(* IEC 61131-3 sources: AXOpen/src/template.axolibrary/ctrl/src/TemplateComponent (part 3) *)

                    IF TRUE THEN
                        THIS.CallTimers(FALSE);
                        _progress := 388;
                    END_IF;
                END_IF;

                IF _progress = 388 THEN                                                                                     // TemplateTask_20steps_2 running: , add_the_detailed_description_of_the_current_action_9
                    IF _infoTimer.output THEN
                        TaskMessenger.Activate( UINT#588, eAxoMessageCategory#Warning);
                        Status.Error.Id :=      UINT#588;
                    END_IF;

                    IF TRUE THEN
                        THIS.CallTimers(FALSE);
                        _progress := 389;
                    END_IF;
                END_IF;

                IF _progress = 389 THEN                                                                                     // TemplateTask_20steps_2 running: , add_the_detailed_description_of_the_current_action_10
                    IF _infoTimer.output THEN
                        TaskMessenger.Activate( UINT#589, eAxoMessageCategory#Warning);
                        Status.Error.Id :=      UINT#589;
                    END_IF;

                    IF TRUE THEN
                        THIS.CallTimers(FALSE);
                        _progress := 390;
                    END_IF;
                END_IF;

                IF _progress = 390 THEN                                                                                     // TemplateTask_20steps_2 running: , add_the_detailed_description_of_the_current_action_11
                    IF _infoTimer.output THEN
                        TaskMessenger.Activate( UINT#590, eAxoMessageCategory#Warning);
                        Status.Error.Id :=      UINT#590;
                    END_IF;

                    IF TRUE THEN
                        THIS.CallTimers(FALSE);
                        _progress := 391;
                    END_IF;
                END_IF;

                IF _progress = 391 THEN                                                                                     // TemplateTask_20steps_2 running: , add_the_detailed_description_of_the_current_action_12
                    IF _infoTimer.output THEN
                        TaskMessenger.Activate( UINT#591, eAxoMessageCategory#Warning);
                        Status.Error.Id :=      UINT#591;
                    END_IF;

                    IF TRUE THEN
                        THIS.CallTimers(FALSE);
                        _progress := 392;
                    END_IF;
                END_IF;

                IF _progress = 392 THEN                                                                                     // TemplateTask_20steps_2 running: , add_the_detailed_description_of_the_current_action_13
                    IF _infoTimer.output THEN
                        TaskMessenger.Activate( UINT#592, eAxoMessageCategory#Warning);
                        Status.Error.Id :=      UINT#592;
                    END_IF;;

                    IF TRUE THEN
                        THIS.CallTimers(FALSE);
                        _progress := 393;
                    END_IF;
                END_IF;

                IF _progress = 393 THEN                                                                                     // TemplateTask_20steps_2 running: , add_the_detailed_description_of_the_current_action_14
                    IF _infoTimer.output THEN
                        TaskMessenger.Activate( UINT#593, eAxoMessageCategory#Warning);
                        Status.Error.Id :=      UINT#593;
                    END_IF;

                    IF TRUE THEN
                        THIS.CallTimers(FALSE);
                        _progress := 394;
                    END_IF;
                END_IF;

                IF _progress = 394 THEN                                                                                     // TemplateTask_20steps_2 running: , add_the_detailed_description_of_the_current_action_15
                    IF _infoTimer.output THEN
                        TaskMessenger.Activate( UINT#594, eAxoMessageCategory#Warning);
                        Status.Error.Id :=      UINT#594;
                    END_IF;

                    IF TRUE THEN
                        THIS.CallTimers(FALSE);
                        _progress := 395;
                    END_IF;
                END_IF;

                IF _progress = 395 THEN                                                                                     // TemplateTask_20steps_2 running: , add_the_detailed_description_of_the_current_action_16
                    IF _infoTimer.output THEN
                        TaskMessenger.Activate( UINT#595, eAxoMessageCategory#Warning);
                        Status.Error.Id :=      UINT#595;
                    END_IF;

                    IF TRUE THEN
                        THIS.CallTimers(FALSE);
                        _progress := 396;
                    END_IF;
                END_IF;

                IF _progress = 396 THEN                                                                                     // TemplateTask_20steps_2 running: , add_the_detailed_description_of_the_current_action_17
                    IF _infoTimer.output THEN
                        TaskMessenger.Activate( UINT#596, eAxoMessageCategory#Warning);
                        Status.Error.Id :=      UINT#596;
                    END_IF;

                    IF TRUE THEN
                        THIS.CallTimers(FALSE);
                        _progress := 397;
                    END_IF;
                END_IF;

                IF _progress = 397 THEN                                                                                     // TemplateTask_20steps_2 running: , add_the_detailed_description_of_the_current_action_18
                    IF _infoTimer.output THEN
                        TaskMessenger.Activate( UINT#597, eAxoMessageCategory#Warning);
                        Status.Error.Id :=      UINT#597;
                    END_IF;

                    IF TRUE THEN
                        THIS.CallTimers(FALSE);
                        _progress := 398;
                    END_IF;
                END_IF;

                IF _progress = 398 THEN                                                                                     // TemplateTask_20steps_2 running: , add_the_detailed_description_of_the_current_action_19
                    IF _infoTimer.output THEN
                        TaskMessenger.Activate( UINT#598, eAxoMessageCategory#Warning);
                        Status.Error.Id :=      UINT#598;
                    END_IF;

                    IF TRUE THEN
                        THIS.CallTimers(FALSE);
                        _progress := 399;
                    END_IF;
                END_IF;

                IF _progress = 399 THEN                                                                                     // TemplateTask_20steps_2 running: , add_the_detailed_description_of_the_current_action_20
                    TemplateTask_20steps_2.DoneWhen(TRUE);
                    _progress := 0;
                END_IF;

                THIS.CallTimers(TRUE);
                TemplateTask_20steps_2.ThrowWhen(_errorTimer.output);
                Status.Action.Id := TO_UINT(_progress);
                TemplateTask_20steps_2.ThrowWhen(TemplateTask_20steps_2.Duration >= Config.TaskTimeout AND Config.TaskTimeout > T#0s ,'TemplateTask_20steps_2 timeout.');
            END_IF;
            IF TemplateTask_20steps_2.DoneReached() THEN
                Status.Action.Id :=  UINT#181;
                Status.Error.Id :=  UINT#0;
            ELSIF TemplateTask_20steps_2.ErrorOccured() THEN
                Status.Action.Id :=  UINT#10080;
                Status.Error.Id  :=  UINT#10080;
            ELSIF TemplateTask_20steps_2.AbortTriggered()THEN
                Status.Action.Id :=  UINT#10081;
                Status.Error.Id  :=  UINT#10081;
            END_IF;
            Messenger.ActivateOnCondition(ULINT#10080,TemplateTask_20steps_2.HasError(), eAxoMessageCategory#Error);
            Messenger.ActivateOnCondition(ULINT#10081,TemplateTask_20steps_2.IsAborted(), eAxoMessageCategory#Error);
            Messenger.ActivateOnCondition(ULINT#182,TemplateTask_20steps_2.RestoreTriggered() , eAxoMessageCategory#Error);
            IF TemplateTask_20steps_2.RestoreTriggered() AND _progress >= 380 AND _progress <= 399  THEN
                Status.Action.Id :=  UINT#182;
                _progress := 0;
            END_IF;
            //**************************************************

            //*************TemplateTask_20steps_3***************
            TemplateTask_20steps_3.SetIsDisabled(FALSE);
            IF TemplateTask_20steps_3.StartTriggered() THEN
                Status.Action.Id :=  UINT#200;
            END_IF;
            Messenger.ActivateOnCondition(ULINT#200,TemplateTask_20steps_3.IsBusy(), eAxoMessageCategory#Info);
            Messenger.ActivateOnCondition(ULINT#201,TemplateTask_20steps_3.IsDone(), eAxoMessageCategory#Info);
            IF TemplateTask_20steps_3.Execute(THIS) THEN
                IF _progress = 0 THEN
                    Status.Error.Id := UINT#0;
                    TaskMessenger.Restore();
                    THIS.CallTimers(FALSE);
                    _progress := 400;
                END_IF;

                IF _progress = 400 THEN                                                                                     // TemplateTask_20steps_3 running: , add_the_detailed_description_of_the_current_action_1
                    IF _infoTimer.output THEN
                        TaskMessenger.Activate( UINT#600, eAxoMessageCategory#Warning);
                        Status.Error.Id :=      UINT#600;
                    END_IF;

                    IF TRUE THEN
                        THIS.CallTimers(FALSE);
                        _progress := 401;
                    END_IF;
                END_IF;

                IF _progress = 401 THEN                                                                                     // TemplateTask_20steps_3 running: , add_the_detailed_description_of_the_current_action_2
                    IF _infoTimer.output THEN
                        TaskMessenger.Activate( UINT#601, eAxoMessageCategory#Warning);
                        Status.Error.Id :=      UINT#601;
                    END_IF;

                    IF TRUE THEN
                        THIS.CallTimers(FALSE);
                        _progress := 402;
                    END_IF;
                END_IF;

                IF _progress = 402 THEN                                                                                     // TemplateTask_20steps_3 running: , add_the_detailed_description_of_the_current_action_3
                    IF _infoTimer.output THEN
                        TaskMessenger.Activate( UINT#602, eAxoMessageCategory#Warning);
                        Status.Error.Id :=      UINT#602;
                    END_IF;

                    IF TRUE THEN
                        THIS.CallTimers(FALSE);
                        _progress := 403;
                    END_IF;
                END_IF;

                IF _progress = 403 THEN                                                                                     // TemplateTask_20steps_3 running: , add_the_detailed_description_of_the_current_action_4
                    IF _infoTimer.output THEN
                        TaskMessenger.Activate( UINT#603, eAxoMessageCategory#Warning);
                        Status.Error.Id :=      UINT#603;
                    END_IF;

                    IF TRUE THEN
                        THIS.CallTimers(FALSE);
                        _progress := 404;
                    END_IF;
                END_IF;

                IF _progress = 404 THEN                                                                                     // TemplateTask_20steps_3 running: , add_the_detailed_description_of_the_current_action_5
                    IF _infoTimer.output THEN
                        TaskMessenger.Activate( UINT#604, eAxoMessageCategory#Warning);
                        Status.Error.Id :=      UINT#604;
                    END_IF;

                    IF TRUE THEN
                        THIS.CallTimers(FALSE);
                        _progress := 405;
                    END_IF;
                END_IF;

                IF _progress = 405 THEN                                                                                     // TemplateTask_20steps_3 running: , add_the_detailed_description_of_the_current_action_6
                    IF _infoTimer.output THEN
                        TaskMessenger.Activate( UINT#605, eAxoMessageCategory#Warning);
                        Status.Error.Id :=      UINT#605;
                    END_IF;

                    IF TRUE THEN
                        THIS.CallTimers(FALSE);
                        _progress := 406;
                    END_IF;
                END_IF;

                IF _progress = 406 THEN                                                                                     // TemplateTask_20steps_3 running: , add_the_detailed_description_of_the_current_action_7
                    IF _infoTimer.output THEN
                        TaskMessenger.Activate( UINT#606, eAxoMessageCategory#Warning);
                        Status.Error.Id :=      UINT#606;
                    END_IF;

                    IF TRUE THEN
                        THIS.CallTimers(FALSE);
                        _progress := 407;
                    END_IF;
                END_IF;

                IF _progress = 407 THEN                                                                                     // TemplateTask_20steps_3 running: , add_the_detailed_description_of_the_current_action_8
                    IF _infoTimer.output THEN
                        TaskMessenger.Activate( UINT#607, eAxoMessageCategory#Warning);
                        Status.Error.Id :=      UINT#607;
                    END_IF;

                    IF TRUE THEN
                        THIS.CallTimers(FALSE);
                        _progress := 408;
                    END_IF;
                END_IF;

                IF _progress = 408 THEN                                                                                     // TemplateTask_20steps_3 running: , add_the_detailed_description_of_the_current_action_9
                    IF _infoTimer.output THEN
                        TaskMessenger.Activate( UINT#608, eAxoMessageCategory#Warning);
                        Status.Error.Id :=      UINT#608;
                    END_IF;

                    IF TRUE THEN
                        THIS.CallTimers(FALSE);
                        _progress := 409;
                    END_IF;
                END_IF;

                IF _progress = 409 THEN                                                                                     // TemplateTask_20steps_3 running: , add_the_detailed_description_of_the_current_action_10
                    IF _infoTimer.output THEN
                        TaskMessenger.Activate( UINT#609, eAxoMessageCategory#Warning);
                        Status.Error.Id :=      UINT#609;
                    END_IF;

                    IF TRUE THEN
                        THIS.CallTimers(FALSE);
                        _progress := 410;
                    END_IF;
                END_IF;

                IF _progress = 410 THEN                                                                                     // TemplateTask_20steps_3 running: , add_the_detailed_description_of_the_current_action_11
                    IF _infoTimer.output THEN
                        TaskMessenger.Activate( UINT#610, eAxoMessageCategory#Warning);
                        Status.Error.Id :=      UINT#610;
                    END_IF;

                    IF TRUE THEN
                        THIS.CallTimers(FALSE);
                        _progress := 411;
                    END_IF;
                END_IF;

                IF _progress = 411 THEN                                                                                     // TemplateTask_20steps_3 running: , add_the_detailed_description_of_the_current_action_12
                    IF _infoTimer.output THEN
                        TaskMessenger.Activate( UINT#611, eAxoMessageCategory#Warning);
                        Status.Error.Id :=      UINT#611;
                    END_IF;

                    IF TRUE THEN
                        THIS.CallTimers(FALSE);
                        _progress := 412;
                    END_IF;
                END_IF;

                IF _progress = 412 THEN                                                                                     // TemplateTask_20steps_3 running: , add_the_detailed_description_of_the_current_action_13
                    IF _infoTimer.output THEN
                        TaskMessenger.Activate( UINT#612, eAxoMessageCategory#Warning);
                        Status.Error.Id :=      UINT#612;
                    END_IF;

                    IF TRUE THEN
                        THIS.CallTimers(FALSE);
                        _progress := 413;
                    END_IF;
                END_IF;

                IF _progress = 413 THEN                                                                                     // TemplateTask_20steps_3 running: , add_the_detailed_description_of_the_current_action_14
                    IF _infoTimer.output THEN
                        TaskMessenger.Activate( UINT#613, eAxoMessageCategory#Warning);
                        Status.Error.Id :=      UINT#613;
                    END_IF;

                    IF TRUE THEN
                        THIS.CallTimers(FALSE);
                        _progress := 414;
                    END_IF;
                END_IF;

                IF _progress = 414 THEN                                                                                     // TemplateTask_20steps_3 running: , add_the_detailed_description_of_the_current_action_15
                    IF _infoTimer.output THEN
                        TaskMessenger.Activate( UINT#614, eAxoMessageCategory#Warning);
                        Status.Error.Id :=      UINT#614;
                    END_IF;

                    IF TRUE THEN
                        THIS.CallTimers(FALSE);
                        _progress := 415;
                    END_IF;
                END_IF;

                IF _progress = 415 THEN                                                                                     // TemplateTask_20steps_3 running: , add_the_detailed_description_of_the_current_action_16
                    IF _infoTimer.output THEN
                        TaskMessenger.Activate( UINT#615, eAxoMessageCategory#Warning);
                        Status.Error.Id :=      UINT#615;
                    END_IF;

                    IF TRUE THEN
                        THIS.CallTimers(FALSE);
                        _progress := 416;
                    END_IF;
                END_IF;

                IF _progress = 416 THEN                                                                                     // TemplateTask_20steps_3 running: , add_the_detailed_description_of_the_current_action_17
                    IF _infoTimer.output THEN
                        TaskMessenger.Activate( UINT#616, eAxoMessageCategory#Warning);
                        Status.Error.Id :=      UINT#616;
                    END_IF;

                    IF TRUE THEN
                        THIS.CallTimers(FALSE);
                        _progress := 417;
                    END_IF;
                END_IF;

                IF _progress = 417 THEN                                                                                     // TemplateTask_20steps_3 running: , add_the_detailed_description_of_the_current_action_18
                    IF _infoTimer.output THEN
                        TaskMessenger.Activate( UINT#617, eAxoMessageCategory#Warning);
                        Status.Error.Id :=      UINT#617;
                    END_IF;

                    IF TRUE THEN
                        THIS.CallTimers(FALSE);
                        _progress := 418;
                    END_IF;
                END_IF;

                IF _progress = 418 THEN                                                                                     // TemplateTask_20steps_3 running: , add_the_detailed_description_of_the_current_action_19
                    IF _infoTimer.output THEN
                        TaskMessenger.Activate( UINT#618, eAxoMessageCategory#Warning);
                        Status.Error.Id :=      UINT#618;
                    END_IF;

                    IF TRUE THEN
                        THIS.CallTimers(FALSE);
                        _progress := 419;
                    END_IF;
                END_IF;

                IF _progress = 419 THEN                                                                                     // TemplateTask_20steps_3 running: , add_the_detailed_description_of_the_current_action_20
                    TemplateTask_20steps_3.DoneWhen(TRUE);
                    _progress := 0;
                END_IF;

                THIS.CallTimers(TRUE);

                TemplateTask_20steps_3.ThrowWhen(_errorTimer.output);
                Status.Action.Id := TO_UINT(_progress);
                TemplateTask_20steps_3.ThrowWhen(TemplateTask_20steps_3.Duration >= Config.TaskTimeout AND Config.TaskTimeout > T#0s ,'TemplateTask_20steps_3 timeout.');
            END_IF;
            IF TemplateTask_20steps_3.DoneReached() THEN
                Status.Action.Id :=  UINT#201;
                Status.Error.Id :=  UINT#0;
            ELSIF TemplateTask_20steps_3.ErrorOccured() THEN
                Status.Action.Id :=  UINT#10100;
                Status.Error.Id  :=  UINT#10100;
            ELSIF TemplateTask_20steps_3.AbortTriggered()THEN
                Status.Action.Id :=  UINT#10101;
                Status.Error.Id  :=  UINT#10101;
            END_IF;
            Messenger.ActivateOnCondition(ULINT#10100,TemplateTask_20steps_3.HasError(), eAxoMessageCategory#Error);
            Messenger.ActivateOnCondition(ULINT#10101,TemplateTask_20steps_3.IsAborted(), eAxoMessageCategory#Error);
            Messenger.ActivateOnCondition(ULINT#202,TemplateTask_20steps_3.RestoreTriggered() , eAxoMessageCategory#Error);
            IF TemplateTask_20steps_3.RestoreTriggered() AND _progress >= 400 AND _progress <= 419  THEN
                Status.Action.Id :=  UINT#202;
                _progress := 0;
            END_IF;
            //**************************************************

            //*************TemplateTask_20steps_4***************
            TemplateTask_20steps_4.SetIsDisabled(FALSE);
            IF TemplateTask_20steps_4.StartTriggered() THEN
                Status.Action.Id :=  UINT#220;
            END_IF;
            Messenger.ActivateOnCondition(ULINT#220,TemplateTask_20steps_4.IsBusy(), eAxoMessageCategory#Info);
            Messenger.ActivateOnCondition(ULINT#221,TemplateTask_20steps_4.IsDone(), eAxoMessageCategory#Info);
            IF TemplateTask_20steps_4.Execute(THIS) THEN
                IF _progress = 0 THEN
                    Status.Error.Id := UINT#0;
                    TaskMessenger.Restore();
                    THIS.CallTimers(FALSE);
                    _progress := 420;
                END_IF;

                IF _progress = 420 THEN                                                                                     // TemplateTask_20steps_4 running: , add_the_detailed_description_of_the_current_action_1
                    IF _infoTimer.output THEN
                        TaskMessenger.Activate( UINT#620, eAxoMessageCategory#Warning);
                        Status.Error.Id :=      UINT#620;
                    END_IF;

                    IF TRUE THEN
                        THIS.CallTimers(FALSE);
                        _progress := 421;
                    END_IF;
                END_IF;

                IF _progress = 421 THEN                                                                                     // TemplateTask_20steps_4 running: , add_the_detailed_description_of_the_current_action_2
                    IF _infoTimer.output THEN
                        TaskMessenger.Activate( UINT#621, eAxoMessageCategory#Warning);
                        Status.Error.Id :=      UINT#621;
                    END_IF;

                    IF TRUE THEN
                        THIS.CallTimers(FALSE);
                        _progress := 422;
                    END_IF;
                END_IF;

                IF _progress = 422 THEN                                                                                     // TemplateTask_20steps_4 running: , add_the_detailed_description_of_the_current_action_3
                    IF _infoTimer.output THEN
                        TaskMessenger.Activate( UINT#622, eAxoMessageCategory#Warning);
                        Status.Error.Id :=      UINT#622;
                    END_IF;

                    IF TRUE THEN
                        THIS.CallTimers(FALSE);
                        _progress := 423;
                    END_IF;
                END_IF;

                IF _progress = 423 THEN                                                                                     // TemplateTask_20steps_4 running: , add_the_detailed_description_of_the_current_action_4
                    IF _infoTimer.output THEN
                        TaskMessenger.Activate( UINT#623, eAxoMessageCategory#Warning);
                        Status.Error.Id :=      UINT#623;
                    END_IF;

                    IF TRUE THEN
                        THIS.CallTimers(FALSE);
                        _progress := 424;
                    END_IF;
                END_IF;

                IF _progress = 424 THEN                                                                                     // TemplateTask_20steps_4 running: , add_the_detailed_description_of_the_current_action_5
                    IF _infoTimer.output THEN
                        TaskMessenger.Activate( UINT#624, eAxoMessageCategory#Warning);
                        Status.Error.Id :=      UINT#624;
                    END_IF;

                    IF TRUE THEN
                        THIS.CallTimers(FALSE);
                        _progress := 425;
                    END_IF;
                END_IF;

                IF _progress = 425 THEN                                                                                     // TemplateTask_20steps_4 running: , add_the_detailed_description_of_the_current_action_6
                    IF _infoTimer.output THEN
                        TaskMessenger.Activate( UINT#625, eAxoMessageCategory#Warning);
                        Status.Error.Id :=      UINT#625;
                    END_IF;

                    IF TRUE THEN
                        THIS.CallTimers(FALSE);
                        _progress := 426;
                    END_IF;
                END_IF;

                IF _progress = 426 THEN                                                                                     // TemplateTask_20steps_4 running: , add_the_detailed_description_of_the_current_action_7
                    IF _infoTimer.output THEN
                        TaskMessenger.Activate( UINT#626, eAxoMessageCategory#Warning);
                        Status.Error.Id :=      UINT#626;
                    END_IF;

                    IF TRUE THEN
                        THIS.CallTimers(FALSE);
                        _progress := 427;
                    END_IF;
                END_IF;

                IF _progress = 427 THEN                                                                                     // TemplateTask_20steps_4 running: , add_the_detailed_description_of_the_current_action_8
                    IF _infoTimer.output THEN
                        TaskMessenger.Activate( UINT#627, eAxoMessageCategory#Warning);
                        Status.Error.Id :=      UINT#627;
                    END_IF;

                    IF TRUE THEN
                        THIS.CallTimers(FALSE);
                        _progress := 428;
                    END_IF;
                END_IF;

                IF _progress = 428 THEN                                                                                     // TemplateTask_20steps_4 running: , add_the_detailed_description_of_the_current_action_9
                    IF _infoTimer.output THEN
                        TaskMessenger.Activate( UINT#628, eAxoMessageCategory#Warning);
                        Status.Error.Id :=      UINT#628;
                    END_IF;

                    IF TRUE THEN
                        THIS.CallTimers(FALSE);
                        _progress := 429;
                    END_IF;
                END_IF;

                IF _progress = 429 THEN                                                                                     // TemplateTask_20steps_4 running: , add_the_detailed_description_of_the_current_action_10
                    IF _infoTimer.output THEN
                        TaskMessenger.Activate( UINT#629, eAxoMessageCategory#Warning);
                        Status.Error.Id :=      UINT#629;
                    END_IF;

                    IF TRUE THEN
                        THIS.CallTimers(FALSE);
                        _progress := 430;
                    END_IF;
                END_IF;

                IF _progress = 430 THEN                                                                                     // TemplateTask_20steps_4 running: , add_the_detailed_description_of_the_current_action_11
                    IF _infoTimer.output THEN
                        TaskMessenger.Activate( UINT#630, eAxoMessageCategory#Warning);
                        Status.Error.Id :=      UINT#630;
                    END_IF;

                    IF TRUE THEN
                        THIS.CallTimers(FALSE);
                        _progress := 431;
                    END_IF;
                END_IF;

                IF _progress = 431 THEN                                                                                     // TemplateTask_20steps_4 running: , add_the_detailed_description_of_the_current_action_12
                    IF _infoTimer.output THEN
                        TaskMessenger.Activate( UINT#631, eAxoMessageCategory#Warning);
                        Status.Error.Id :=      UINT#631;
                    END_IF;

                    IF TRUE THEN
                        THIS.CallTimers(FALSE);
                        _progress := 432;
                    END_IF;
                END_IF;

                IF _progress = 432 THEN                                                                                     // TemplateTask_20steps_4 running: , add_the_detailed_description_of_the_current_action_13
                    IF _infoTimer.output THEN
                        TaskMessenger.Activate( UINT#632, eAxoMessageCategory#Warning);
                        Status.Error.Id :=      UINT#632;
                    END_IF;

                    IF TRUE THEN
                        THIS.CallTimers(FALSE);
                        _progress := 433;
                    END_IF;
                END_IF;

                IF _progress = 433 THEN                                                                                     // TemplateTask_20steps_4 running: , add_the_detailed_description_of_the_current_action_14
                    IF _infoTimer.output THEN
                        TaskMessenger.Activate( UINT#633, eAxoMessageCategory#Warning);
                        Status.Error.Id :=      UINT#633;
                    END_IF;

                    IF TRUE THEN
                        THIS.CallTimers(FALSE);
                        _progress := 434;
                    END_IF;
                END_IF;

                IF _progress = 434 THEN                                                                                     // TemplateTask_20steps_4 running: , add_the_detailed_description_of_the_current_action_15
                    IF _infoTimer.output THEN
                        TaskMessenger.Activate( UINT#634, eAxoMessageCategory#Warning);
                        Status.Error.Id :=      UINT#634;
                    END_IF;

                    IF TRUE THEN
                        THIS.CallTimers(FALSE);
                        _progress := 435;
                    END_IF;
                END_IF;

                IF _progress = 435 THEN                                                                                     // TemplateTask_20steps_4 running: , add_the_detailed_description_of_the_current_action_16
                    IF _infoTimer.output THEN
                        TaskMessenger.Activate( UINT#635, eAxoMessageCategory#Warning);
                        Status.Error.Id :=      UINT#635;
                    END_IF;

                    IF TRUE THEN
                        THIS.CallTimers(FALSE);
                        _progress := 436;
                    END_IF;
                END_IF;

                IF _progress = 436 THEN                                                                                     // TemplateTask_20steps_4 running: , add_the_detailed_description_of_the_current_action_17
                    IF _infoTimer.output THEN
                        TaskMessenger.Activate( UINT#636, eAxoMessageCategory#Warning);
                        Status.Error.Id :=      UINT#636;
                    END_IF;

                    IF TRUE THEN
                        THIS.CallTimers(FALSE);
                        _progress := 437;
                    END_IF;
                END_IF;

                IF _progress = 437 THEN                                                                                     // TemplateTask_20steps_4 running: , add_the_detailed_description_of_the_current_action_18
                    IF _infoTimer.output THEN
                        TaskMessenger.Activate( UINT#637, eAxoMessageCategory#Warning);
                        Status.Error.Id :=      UINT#637;
                    END_IF;

                    IF TRUE THEN
                        THIS.CallTimers(FALSE);
                        _progress := 438;
                    END_IF;
                END_IF;

                IF _progress = 438 THEN                                                                                     // TemplateTask_20steps_4 running: , add_the_detailed_description_of_the_current_action_19
                    IF _infoTimer.output THEN
                        TaskMessenger.Activate( UINT#638, eAxoMessageCategory#Warning);
                        Status.Error.Id :=      UINT#638;
                    END_IF;

                    IF TRUE THEN
                        THIS.CallTimers(FALSE);
                        _progress := 439;
                    END_IF;
                END_IF;

                IF _progress = 439 THEN                                                                                     // TemplateTask_20steps_4 running: , add_the_detailed_description_of_the_current_action_20
                    TemplateTask_20steps_4.DoneWhen(TRUE);
                    _progress := 0;
                END_IF;

                THIS.CallTimers(TRUE);

                TemplateTask_20steps_4.ThrowWhen(_errorTimer.output);
                Status.Action.Id := TO_UINT(_progress);
                TemplateTask_20steps_4.ThrowWhen(TemplateTask_20steps_4.Duration >= Config.TaskTimeout AND Config.TaskTimeout > T#0s ,'TemplateTask_20steps_4 timeout.');
            END_IF;
            IF TemplateTask_20steps_4.DoneReached() THEN
                Status.Action.Id :=  UINT#221;
                Status.Error.Id :=  UINT#0;
            ELSIF TemplateTask_20steps_4.ErrorOccured() THEN
                Status.Action.Id :=  UINT#10120;
                Status.Error.Id  :=  UINT#10120;
            ELSIF TemplateTask_20steps_4.AbortTriggered()THEN
                Status.Action.Id :=  UINT#10121;
                Status.Error.Id  :=  UINT#10121;
            END_IF;
            Messenger.ActivateOnCondition(ULINT#10120,TemplateTask_20steps_4.HasError(), eAxoMessageCategory#Error);
            Messenger.ActivateOnCondition(ULINT#10121,TemplateTask_20steps_4.IsAborted(), eAxoMessageCategory#Error);
            Messenger.ActivateOnCondition(ULINT#222,TemplateTask_20steps_4.RestoreTriggered() , eAxoMessageCategory#Error);
            IF TemplateTask_20steps_4.RestoreTriggered() AND _progress >= 420 AND _progress <= 439  THEN
                Status.Action.Id :=  UINT#222;
                _progress := 0;
            END_IF;
            //**************************************************

            //*************TemplateTask_20steps_5***************
            TemplateTask_20steps_5.SetIsDisabled(FALSE);
            IF TemplateTask_20steps_5.StartTriggered() THEN
                Status.Action.Id :=  UINT#240;
            END_IF;
            Messenger.ActivateOnCondition(ULINT#240,TemplateTask_20steps_5.IsBusy(), eAxoMessageCategory#Info);
            Messenger.ActivateOnCondition(ULINT#241,TemplateTask_20steps_5.IsDone(), eAxoMessageCategory#Info);
            IF TemplateTask_20steps_5.Execute(THIS) THEN
                IF _progress = 0 THEN
                    Status.Error.Id := UINT#0;
                    TaskMessenger.Restore();
                    THIS.CallTimers(FALSE);
                    _progress := 440;
                END_IF;

                IF _progress = 440 THEN                                                                                     // TemplateTask_20steps_5 running: , add_the_detailed_description_of_the_current_action_1
                    IF _infoTimer.output THEN
                        TaskMessenger.Activate( UINT#640, eAxoMessageCategory#Warning);
                        Status.Error.Id :=      UINT#640;
                    END_IF;

                    IF TRUE THEN
                        THIS.CallTimers(FALSE);
                        _progress := 441;
                    END_IF;
                END_IF;

                IF _progress = 441 THEN                                                                                     // TemplateTask_20steps_5 running , add_the_detailed_description_of_the_current_action_2
                    IF _infoTimer.output THEN
                        TaskMessenger.Activate( UINT#641, eAxoMessageCategory#Warning);
                        Status.Error.Id :=      UINT#641;
                    END_IF;

                    IF TRUE THEN
                        THIS.CallTimers(FALSE);
                        _progress := 442;
                    END_IF;
                END_IF;

                IF _progress = 442 THEN                                                                                     // TemplateTask_20steps_5 running: , add_the_detailed_description_of_the_current_action_3
                    IF _infoTimer.output THEN
                        TaskMessenger.Activate( UINT#642, eAxoMessageCategory#Warning);
                        Status.Error.Id :=      UINT#642;
                    END_IF;

                    IF TRUE THEN
                        THIS.CallTimers(FALSE);
                        _progress := 443;
                    END_IF;
                END_IF;

                IF _progress = 443 THEN                                                                                     // TemplateTask_20steps_5 running: , add_the_detailed_description_of_the_current_action_4
                    IF _infoTimer.output THEN
                        TaskMessenger.Activate( UINT#643, eAxoMessageCategory#Warning);
                        Status.Error.Id :=      UINT#643;
                    END_IF;

                    IF TRUE THEN
                        THIS.CallTimers(FALSE);
                        _progress := 444;
                    END_IF;
                END_IF;

                IF _progress = 444 THEN                                                                                     // TemplateTask_20steps_5 running: , add_the_detailed_description_of_the_current_action_5
                    IF _infoTimer.output THEN
                        TaskMessenger.Activate( UINT#644, eAxoMessageCategory#Warning);
                        Status.Error.Id :=      UINT#644;
                    END_IF;

                    IF TRUE THEN
                        THIS.CallTimers(FALSE);
                        _progress := 445;
                    END_IF;
                END_IF;

                IF _progress = 445 THEN                                                                                     // TemplateTask_20steps_5 running: , add_the_detailed_description_of_the_current_action_6
                    IF _infoTimer.output THEN
                        TaskMessenger.Activate( UINT#645, eAxoMessageCategory#Warning);
                        Status.Error.Id :=      UINT#645;
                    END_IF;

                    IF TRUE THEN
                        THIS.CallTimers(FALSE);
                        _progress := 446;
                    END_IF;
                END_IF;

                IF _progress = 446 THEN                                                                                     // TemplateTask_20steps_5 running: , add_the_detailed_description_of_the_current_action_7
                    IF _infoTimer.output THEN
                        TaskMessenger.Activate( UINT#646, eAxoMessageCategory#Warning);
                        Status.Error.Id :=      UINT#646;
                    END_IF;

                    IF TRUE THEN
                        THIS.CallTimers(FALSE);
                        _progress := 447;
                    END_IF;
                END_IF;

                IF _progress = 447 THEN                                                                                     // TemplateTask_20steps_5 running: , add_the_detailed_description_of_the_current_action_8
                    IF _infoTimer.output THEN
                        TaskMessenger.Activate( UINT#647, eAxoMessageCategory#Warning);
                        Status.Error.Id :=      UINT#647;
                    END_IF;

                    IF TRUE THEN
                        THIS.CallTimers(FALSE);
                        _progress := 448;
                    END_IF;
                END_IF;

                IF _progress = 448 THEN                                                                                     // TemplateTask_20steps_5 running: , add_the_detailed_description_of_the_current_action_9
                    IF _infoTimer.output THEN
                        TaskMessenger.Activate( UINT#648, eAxoMessageCategory#Warning);
                        Status.Error.Id :=      UINT#648;
                    END_IF;

                    IF TRUE THEN
                        THIS.CallTimers(FALSE);
                        _progress := 449;
                    END_IF;
                END_IF;

                IF _progress = 449 THEN                                                                                     // TemplateTask_20steps_5 running: , add_the_detailed_description_of_the_current_action_10
                    IF _infoTimer.output THEN
                        TaskMessenger.Activate( UINT#649, eAxoMessageCategory#Warning);
                        Status.Error.Id :=      UINT#649;
                    END_IF;

                    IF TRUE THEN
                        THIS.CallTimers(FALSE);
                        _progress := 450;
                    END_IF;
                END_IF;

                IF _progress = 450 THEN                                                                                     // TemplateTask_20steps_5 running: , add_the_detailed_description_of_the_current_action_11
                    IF _infoTimer.output THEN
                        TaskMessenger.Activate( UINT#650, eAxoMessageCategory#Warning);
                        Status.Error.Id :=      UINT#650;
                    END_IF;

                    IF TRUE THEN
                        THIS.CallTimers(FALSE);
                        _progress := 451;
                    END_IF;
                END_IF;

                IF _progress = 451 THEN                                                                                     // TemplateTask_20steps_5 running: , add_the_detailed_description_of_the_current_action_12
                    IF _infoTimer.output THEN
                        TaskMessenger.Activate( UINT#651, eAxoMessageCategory#Warning);
                        Status.Error.Id :=      UINT#651;
                    END_IF;

                    IF TRUE THEN
                        THIS.CallTimers(FALSE);
                        _progress := 452;
                    END_IF;
                END_IF;

                IF _progress = 452 THEN                                                                                     // TemplateTask_20steps_5 running: , add_the_detailed_description_of_the_current_action_13
                    IF _infoTimer.output THEN
                        TaskMessenger.Activate( UINT#652, eAxoMessageCategory#Warning);
                        Status.Error.Id :=      UINT#652;
                    END_IF;

                    IF TRUE THEN
                        THIS.CallTimers(FALSE);
                        _progress := 453;
                    END_IF;
                END_IF;

                IF _progress = 453 THEN                                                                                     // TemplateTask_20steps_5 running: , add_the_detailed_description_of_the_current_action_14
                    IF _infoTimer.output THEN
                        TaskMessenger.Activate( UINT#653, eAxoMessageCategory#Warning);
                        Status.Error.Id :=      UINT#653;
                    END_IF;

                    IF TRUE THEN
                        THIS.CallTimers(FALSE);
                        _progress := 454;
                    END_IF;
                END_IF;

                IF _progress = 454 THEN                                                                                     // TemplateTask_20steps_5 running: , add_the_detailed_description_of_the_current_action_15
                    IF _infoTimer.output THEN
                        TaskMessenger.Activate( UINT#654, eAxoMessageCategory#Warning);
                        Status.Error.Id :=      UINT#654;
                    END_IF;

                    IF TRUE THEN
                        THIS.CallTimers(FALSE);
                        _progress := 455;
                    END_IF;
                END_IF;

                IF _progress = 455 THEN                                                                                     // TemplateTask_20steps_5 running: , add_the_detailed_description_of_the_current_action_16
                    IF _infoTimer.output THEN
                        TaskMessenger.Activate( UINT#655, eAxoMessageCategory#Warning);
                        Status.Error.Id :=      UINT#655;
                    END_IF;

                    IF TRUE THEN
                        THIS.CallTimers(FALSE);
                        _progress := 456;
                    END_IF;
                END_IF;

                IF _progress = 456 THEN                                                                                     // TemplateTask_20steps_5 running: , add_the_detailed_description_of_the_current_action_17
                    IF _infoTimer.output THEN
                        TaskMessenger.Activate( UINT#656, eAxoMessageCategory#Warning);
                        Status.Error.Id :=      UINT#656;
                    END_IF;

                    IF TRUE THEN
                        THIS.CallTimers(FALSE);
                        _progress := 457;
                    END_IF;
                END_IF;

                IF _progress = 457 THEN                                                                                     // TemplateTask_20steps_5 running: , add_the_detailed_description_of_the_current_action_18
                    IF _infoTimer.output THEN
                        TaskMessenger.Activate( UINT#657, eAxoMessageCategory#Warning);
                        Status.Error.Id :=      UINT#657;
                    END_IF;

                    IF TRUE THEN
                        THIS.CallTimers(FALSE);
                        _progress := 458;
                    END_IF;
                END_IF;

                IF _progress = 458 THEN                                                                                     // TemplateTask_20steps_5 running: , add_the_detailed_description_of_the_current_action_19
                    IF _infoTimer.output THEN
                        TaskMessenger.Activate( UINT#658, eAxoMessageCategory#Warning);
                        Status.Error.Id :=      UINT#658;
                    END_IF;

                    IF TRUE THEN
                        THIS.CallTimers(FALSE);
                        _progress := 459;
                    END_IF;
                END_IF;

                IF _progress = 459 THEN                                                                                     // TemplateTask_20steps_5 running: , add_the_detailed_description_of_the_current_action_20
                    TemplateTask_20steps_5.DoneWhen(TRUE);
                    _progress := 0;
                END_IF;

                THIS.CallTimers(TRUE);

                TemplateTask_20steps_5.ThrowWhen(_errorTimer.output);
                Status.Action.Id := TO_UINT(_progress);
                TemplateTask_20steps_5.ThrowWhen(TemplateTask_20steps_5.Duration >= Config.TaskTimeout AND Config.TaskTimeout > T#0s ,'TemplateTask_20steps_5 timeout.');
            END_IF;
            IF TemplateTask_20steps_5.DoneReached() THEN
                Status.Action.Id :=  UINT#241;
                Status.Error.Id :=  UINT#0;
            ELSIF TemplateTask_20steps_5.ErrorOccured() THEN
                Status.Action.Id :=  UINT#10140;
                Status.Error.Id  :=  UINT#10140;
            ELSIF TemplateTask_20steps_5.AbortTriggered()THEN
                Status.Action.Id :=  UINT#10141;
                Status.Error.Id  :=  UINT#10141;
            END_IF;
            Messenger.ActivateOnCondition(ULINT#10140,TemplateTask_20steps_5.HasError(), eAxoMessageCategory#Error);
            Messenger.ActivateOnCondition(ULINT#10141,TemplateTask_20steps_5.IsAborted(), eAxoMessageCategory#Error);
            Messenger.ActivateOnCondition(ULINT#242,TemplateTask_20steps_5.RestoreTriggered() , eAxoMessageCategory#Error);
            IF TemplateTask_20steps_5.RestoreTriggered() AND _progress >= 440 AND _progress <= 459  THEN
                Status.Action.Id :=  UINT#242;
                _progress := 0;
            END_IF;
            //**************************************************

            //*************TemplateTask_20steps_6***************
            TemplateTask_20steps_6.SetIsDisabled(FALSE);
            IF TemplateTask_20steps_6.StartTriggered() THEN
                Status.Action.Id :=  UINT#260;
            END_IF;
            Messenger.ActivateOnCondition(ULINT#260,TemplateTask_20steps_6.IsBusy(), eAxoMessageCategory#Info);
            Messenger.ActivateOnCondition(ULINT#261,TemplateTask_20steps_6.IsDone(), eAxoMessageCategory#Info);
            IF TemplateTask_20steps_6.Execute(THIS) THEN
                IF _progress = 0 THEN
                    Status.Error.Id := UINT#0;
                    TaskMessenger.Restore();
                    THIS.CallTimers(FALSE);
                    _progress := 460;
                END_IF;

                IF _progress = 460 THEN                                                                                     // TemplateTask_20steps_6 running: , add_the_detailed_description_of_the_current_action_1
                    IF _infoTimer.output THEN
                        TaskMessenger.Activate( UINT#660, eAxoMessageCategory#Warning);
                        Status.Error.Id :=      UINT#660;
                    END_IF;

                    IF TRUE THEN
                        THIS.CallTimers(FALSE);
                        _progress := 461;
                    END_IF;
                END_IF;

                IF _progress = 461 THEN                                                                                     // TemplateTask_20steps_6 running: , add_the_detailed_description_of_the_current_action_2
                    IF _infoTimer.output THEN
                        TaskMessenger.Activate( UINT#661, eAxoMessageCategory#Warning);
                        Status.Error.Id :=      UINT#661;
                    END_IF;

                    IF TRUE THEN
                        THIS.CallTimers(FALSE);
                        _progress := 462;
                    END_IF;
                END_IF;

                IF _progress = 462 THEN                                                                                     // TemplateTask_20steps_6 running: , add_the_detailed_description_of_the_current_action_3
                    IF _infoTimer.output THEN
                        TaskMessenger.Activate( UINT#662, eAxoMessageCategory#Warning);
                        Status.Error.Id :=      UINT#662;
                    END_IF;

                    IF TRUE THEN
                        THIS.CallTimers(FALSE);
                        _progress := 463;
                    END_IF;
                END_IF;

                IF _progress = 463 THEN                                                                                     // TemplateTask_20steps_6 running: , add_the_detailed_description_of_the_current_action_4
                    IF _infoTimer.output THEN
                        TaskMessenger.Activate( UINT#663, eAxoMessageCategory#Warning);
                        Status.Error.Id :=      UINT#663;
                    END_IF;

                    IF TRUE THEN
                        THIS.CallTimers(FALSE);
                        _progress := 464;
                    END_IF;
                END_IF;

                IF _progress = 464 THEN                                                                                     // TemplateTask_20steps_6 running: , add_the_detailed_description_of_the_current_action_5
                    IF _infoTimer.output THEN
                        TaskMessenger.Activate( UINT#664, eAxoMessageCategory#Warning);
                        Status.Error.Id :=      UINT#664;
                    END_IF;

                    IF TRUE THEN
                        THIS.CallTimers(FALSE);
                        _progress := 465;
                    END_IF;
                END_IF;

                IF _progress = 465 THEN                                                                                     // TemplateTask_20steps_6 running: , add_the_detailed_description_of_the_current_action_6
                    IF _infoTimer.output THEN
                        TaskMessenger.Activate( UINT#665, eAxoMessageCategory#Warning);
                        Status.Error.Id :=      UINT#665;
                    END_IF;

                    IF TRUE THEN
                        THIS.CallTimers(FALSE);
                        _progress := 466;
                    END_IF;
                END_IF;

                IF _progress = 466 THEN                                                                                     // TemplateTask_20steps_6 running: , add_the_detailed_description_of_the_current_action_7
                    IF _infoTimer.output THEN
                        TaskMessenger.Activate( UINT#666, eAxoMessageCategory#Warning);
                        Status.Error.Id :=      UINT#666;
                    END_IF;

                    IF TRUE THEN
                        THIS.CallTimers(FALSE);
                        _progress := 467;
                    END_IF;
                END_IF;

                IF _progress = 467 THEN                                                                                     // TemplateTask_20steps_6 running: , add_the_detailed_description_of_the_current_action_8
                    IF _infoTimer.output THEN
                        TaskMessenger.Activate( UINT#667, eAxoMessageCategory#Warning);
                        Status.Error.Id :=      UINT#667;
                    END_IF;

                    IF TRUE THEN
                        THIS.CallTimers(FALSE);
                        _progress := 468;
                    END_IF;
                END_IF;

                IF _progress = 468 THEN                                                                                     // TemplateTask_20steps_6 running: , add_the_detailed_description_of_the_current_action_9
                    IF _infoTimer.output THEN
                        TaskMessenger.Activate( UINT#668, eAxoMessageCategory#Warning);
                        Status.Error.Id :=      UINT#668;
                    END_IF;

                    IF TRUE THEN
                        THIS.CallTimers(FALSE);
                        _progress := 469;
                    END_IF;
                END_IF;

                IF _progress = 469 THEN                                                                                     // TemplateTask_20steps_6 running: , add_the_detailed_description_of_the_current_action_10
                    IF _infoTimer.output THEN
                        TaskMessenger.Activate( UINT#669, eAxoMessageCategory#Warning);
                        Status.Error.Id :=      UINT#669;
                    END_IF;

                    IF TRUE THEN
                        THIS.CallTimers(FALSE);
                        _progress := 470;
                    END_IF;
                END_IF;

                IF _progress = 470 THEN                                                                                     // TemplateTask_20steps_6 running: , add_the_detailed_description_of_the_current_action_11
                    IF _infoTimer.output THEN
                        TaskMessenger.Activate( UINT#670, eAxoMessageCategory#Warning);
                        Status.Error.Id :=      UINT#670;
                    END_IF;

                    IF TRUE THEN
                        THIS.CallTimers(FALSE);
                        _progress := 471;
                    END_IF;
                END_IF;

                IF _progress = 471 THEN                                                                                     // TemplateTask_20steps_6 running: , add_the_detailed_description_of_the_current_action_12
                    IF _infoTimer.output THEN
                        TaskMessenger.Activate( UINT#671, eAxoMessageCategory#Warning);
                        Status.Error.Id :=      UINT#671;
                    END_IF;

                    IF TRUE THEN
                        THIS.CallTimers(FALSE);
                        _progress := 472;
                    END_IF;
                END_IF;

                IF _progress = 472 THEN                                                                                     // TemplateTask_20steps_6 running: , add_the_detailed_description_of_the_current_action_13
                    IF _infoTimer.output THEN
                        TaskMessenger.Activate( UINT#672, eAxoMessageCategory#Warning);
                        Status.Error.Id :=      UINT#672;
                    END_IF;

                    IF TRUE THEN
                        THIS.CallTimers(FALSE);
                        _progress := 473;
                    END_IF;
                END_IF;

                IF _progress = 473 THEN                                                                                     // TemplateTask_20steps_6 running: , add_the_detailed_description_of_the_current_action_14
                    IF _infoTimer.output THEN
                        TaskMessenger.Activate( UINT#673, eAxoMessageCategory#Warning);
                        Status.Error.Id :=      UINT#673;
                    END_IF;

                    IF TRUE THEN
                        THIS.CallTimers(FALSE);
                        _progress := 474;
                    END_IF;
                END_IF;

                IF _progress = 474 THEN                                                                                     // TemplateTask_20steps_6 running: , add_the_detailed_description_of_the_current_action_15
                    IF _infoTimer.output THEN
                        TaskMessenger.Activate( UINT#674, eAxoMessageCategory#Warning);
                        Status.Error.Id :=      UINT#674;
                    END_IF;

                    IF TRUE THEN
                        THIS.CallTimers(FALSE);
                        _progress := 475;
                    END_IF;
                END_IF;

                IF _progress = 475 THEN                                                                                     // TemplateTask_20steps_6 running: , add_the_detailed_description_of_the_current_action_16
                    IF _infoTimer.output THEN
                        TaskMessenger.Activate( UINT#675, eAxoMessageCategory#Warning);
                        Status.Error.Id :=      UINT#675;
                    END_IF;

                    IF TRUE THEN
                        THIS.CallTimers(FALSE);
                        _progress := 476;
                    END_IF;
                END_IF;

                IF _progress = 476 THEN                                                                                     // TemplateTask_20steps_6 running: , add_the_detailed_description_of_the_current_action_17
                    IF _infoTimer.output THEN
                        TaskMessenger.Activate( UINT#676, eAxoMessageCategory#Warning);
                        Status.Error.Id :=      UINT#676;
                    END_IF;

                    IF TRUE THEN
                        THIS.CallTimers(FALSE);
                        _progress := 477;
                    END_IF;
                END_IF;

                IF _progress = 477 THEN                                                                                     // TemplateTask_20steps_6 running: , add_the_detailed_description_of_the_current_action_18
                    IF _infoTimer.output THEN
                        TaskMessenger.Activate( UINT#677, eAxoMessageCategory#Warning);
                        Status.Error.Id :=      UINT#677;
                    END_IF;

                    IF TRUE THEN
                        THIS.CallTimers(FALSE);
                        _progress := 478;
                    END_IF;
                END_IF;

                IF _progress = 478 THEN                                                                                     // TemplateTask_20steps_6 running: , add_the_detailed_description_of_the_current_action_19
                    IF _infoTimer.output THEN
                        TaskMessenger.Activate( UINT#678, eAxoMessageCategory#Warning);
                        Status.Error.Id :=      UINT#678;
                    END_IF;

                    IF TRUE THEN
                        THIS.CallTimers(FALSE);
                        _progress := 479;
                    END_IF;
                END_IF;

                IF _progress = 479 THEN                                                                                     // TemplateTask_20steps_6 running: , add_the_detailed_description_of_the_current_action_20
                    TemplateTask_20steps_6.DoneWhen(TRUE);
                    _progress := 0;
                END_IF;

                THIS.CallTimers(TRUE);

                TemplateTask_20steps_6.ThrowWhen(_errorTimer.output);
                Status.Action.Id := TO_UINT(_progress);
                TemplateTask_20steps_6.ThrowWhen(TemplateTask_20steps_6.Duration >= Config.TaskTimeout AND Config.TaskTimeout > T#0s ,'TemplateTask_20steps_6 timeout.');
            END_IF;
            IF TemplateTask_20steps_6.DoneReached() THEN
                Status.Action.Id :=  UINT#261;
                Status.Error.Id :=  UINT#0;
            ELSIF TemplateTask_20steps_6.ErrorOccured() THEN
                Status.Action.Id :=  UINT#10160;
                Status.Error.Id  :=  UINT#10160;
            ELSIF TemplateTask_20steps_6.AbortTriggered()THEN
                Status.Action.Id :=  UINT#10161;
                Status.Error.Id  :=  UINT#10161;
            END_IF;
            Messenger.ActivateOnCondition(ULINT#10160,TemplateTask_20steps_6.HasError(), eAxoMessageCategory#Error);
            Messenger.ActivateOnCondition(ULINT#10161,TemplateTask_20steps_6.IsAborted(), eAxoMessageCategory#Error);
            Messenger.ActivateOnCondition(ULINT#262,TemplateTask_20steps_6.RestoreTriggered() , eAxoMessageCategory#Error);
            IF TemplateTask_20steps_6.RestoreTriggered() AND _progress >= 460 AND _progress <= 479  THEN
                Status.Action.Id :=  UINT#262;
                _progress := 0;
            END_IF;
            //******************************************

            //***********Update outputs ****************
            // _data_out_1[0].%X1                  :=      TemplateComponentOutputStructure_hwID_out_1.Item1;
            // _data_out_1[0].%X2                  :=      TemplateComponentOutputStructure_hwID_out_1.Item2;
            // _data_out_1[0].%X3                  :=      TemplateComponentOutputStructure_hwID_out_1.Item1;
            // _data_out_1[0].%X4                  :=      TemplateComponentOutputStructure_hwID_out_1.Item2;

            _retVal := Siemens.Simatic.DistributedIO.WriteData((Config.HWIDs.HwID_out_1),_data_out_1);
            IF _retVal > WORD#0 THEN
                Messenger.Activate(UINT#1231, eAxoMessageCategory#ProgrammingError);
                Status.Error.Id := UINT#1231;
                RETURN;
            END_IF;

            // _data_out_1[0].%X1                  :=      TemplateComponentOutputStructure_hwID_out_2.Item1;
            // _data_out_1[0].%X2                  :=      TemplateComponentOutputStructure_hwID_out_2.Item2;
            // _data_out_1[0].%X3                  :=      TemplateComponentOutputStructure_hwID_out_2.Item1;
            // _data_out_1[0].%X4                  :=      TemplateComponentOutputStructure_hwID_out_2.Item2;

            _retVal := Siemens.Simatic.DistributedIO.WriteData((Config.HWIDs.HwID_out_2),_data_out_1);
            IF _retVal > WORD#0 THEN
                Messenger.Activate(UINT#1232, eAxoMessageCategory#ProgrammingError);
                Status.Error.Id := UINT#1232;
                RETURN;
            END_IF;

            // _data_out_4[1]                     :=      TO_WORD(TemplateComponentOutputStructure_hwID_out_3.Item1).%B0;
            // _data_out_4[0]                     :=      TO_WORD(TemplateComponentOutputStructure_hwID_out_3.Item1).%B1;
            // _data_out_4[3]                     :=      TO_WORD(TemplateComponentOutputStructure_hwID_out_3.Item2).%B0;
            // _data_out_4[2]                     :=      TO_WORD(TemplateComponentOutputStructure_hwID_out_3.Item2).%B1;

            _retVal := Siemens.Simatic.DistributedIO.WriteData((Config.HWIDs.HwID_out_3),_data_out_4);
            IF _retVal > WORD#0 THEN
                Messenger.Activate(UINT#1233, eAxoMessageCategory#ProgrammingError);
                Status.Error.Id := UINT#1233;
                RETURN;
            END_IF;

            // _data_out_8[3]                     :=      TO_DWORD(TemplateComponentOutputStructure_hwID_out_4.Item1).%B0;
            // _data_out_8[2]                     :=      TO_DWORD(TemplateComponentOutputStructure_hwID_out_4.Item1).%B1;
            // _data_out_8[1]                     :=      TO_DWORD(TemplateComponentOutputStructure_hwID_out_4.Item1).%B2;
            // _data_out_8[0]                     :=      TO_DWORD(TemplateComponentOutputStructure_hwID_out_4.Item1).%B3;
            // _data_out_8[7]                     :=      TO_DWORD(TemplateComponentOutputStructure_hwID_out_4.Item2).%B0;
            // _data_out_8[6]                     :=      TO_DWORD(TemplateComponentOutputStructure_hwID_out_4.Item2).%B1;
            // _data_out_8[5]                     :=      TO_DWORD(TemplateComponentOutputStructure_hwID_out_4.Item2).%B2;
            // _data_out_8[4]                     :=      TO_DWORD(TemplateComponentOutputStructure_hwID_out_4.Item2).%B3;

            _retVal := Siemens.Simatic.DistributedIO.WriteData((Config.HWIDs.HwID_out_4),_data_out_8);
            IF _retVal > WORD#0 THEN
                Messenger.Activate(UINT#1234, eAxoMessageCategory#ProgrammingError);
                Status.Error.Id := UINT#1234;
                RETURN;
            END_IF;

            // _data_out_8[3]                     :=      TO_DWORD(TemplateComponentOutputStructure_hwID_out_5.Item1).%B0;
            // _data_out_8[2]                     :=      TO_DWORD(TemplateComponentOutputStructure_hwID_out_5.Item1).%B1;
            // _data_out_8[1]                     :=      TO_DWORD(TemplateComponentOutputStructure_hwID_out_5.Item1).%B2;
            // _data_out_8[0]                     :=      TO_DWORD(TemplateComponentOutputStructure_hwID_out_5.Item1).%B3;
            // _data_out_8[7]                     :=      TO_DWORD(TemplateComponentOutputStructure_hwID_out_5.Item2).%B0;
            // _data_out_8[6]                     :=      TO_DWORD(TemplateComponentOutputStructure_hwID_out_5.Item2).%B1;
            // _data_out_8[5]                     :=      TO_DWORD(TemplateComponentOutputStructure_hwID_out_5.Item2).%B2;
            // _data_out_8[4]                     :=      TO_DWORD(TemplateComponentOutputStructure_hwID_out_5.Item2).%B3;

            _retVal := Siemens.Simatic.DistributedIO.WriteData((Config.HWIDs.HwID_out_5),_data_out_8);
            IF _retVal > WORD#0 THEN
                Messenger.Activate(UINT#1235, eAxoMessageCategory#ProgrammingError);
                Status.Error.Id := UINT#1235;
                RETURN;
            END_IF;

            // _data_out_8[3]                     :=      TO_DWORD(TemplateComponentOutputStructure_hwID_out_6.Item1).%B0;
            // _data_out_8[2]                     :=      TO_DWORD(TemplateComponentOutputStructure_hwID_out_6.Item1).%B1;
            // _data_out_8[1]                     :=      TO_DWORD(TemplateComponentOutputStructure_hwID_out_6.Item1).%B2;
            // _data_out_8[0]                     :=      TO_DWORD(TemplateComponentOutputStructure_hwID_out_6.Item1).%B3;
            // _data_out_8[7]                     :=      TO_DWORD(TemplateComponentOutputStructure_hwID_out_6.Item2).%B0;
            // _data_out_8[6]                     :=      TO_DWORD(TemplateComponentOutputStructure_hwID_out_6.Item2).%B1;
            // _data_out_8[5]                     :=      TO_DWORD(TemplateComponentOutputStructure_hwID_out_6.Item2).%B2;
            // _data_out_8[4]                     :=      TO_DWORD(TemplateComponentOutputStructure_hwID_out_6.Item2).%B3;

            _retVal := Siemens.Simatic.DistributedIO.WriteData((Config.HWIDs.HwID_out_6),_data_out_8);
            IF _retVal > WORD#0 THEN
                Messenger.Activate(UINT#1236, eAxoMessageCategory#ProgrammingError);
                Status.Error.Id := UINT#1236;
                RETURN;
            END_IF;

            // _data_out_8[3]                     :=      TO_DWORD(TemplateComponentOutputStructure_hwID_out_7.Item1).%B0;
            // _data_out_8[2]                     :=      TO_DWORD(TemplateComponentOutputStructure_hwID_out_7.Item1).%B1;
            // _data_out_8[1]                     :=      TO_DWORD(TemplateComponentOutputStructure_hwID_out_7.Item1).%B2;
            // _data_out_8[0]                     :=      TO_DWORD(TemplateComponentOutputStructure_hwID_out_7.Item1).%B3;
            // _data_out_8[7]                     :=      TO_DWORD(TemplateComponentOutputStructure_hwID_out_7.Item2).%B0;
            // _data_out_8[6]                     :=      TO_DWORD(TemplateComponentOutputStructure_hwID_out_7.Item2).%B1;
            // _data_out_8[5]                     :=      TO_DWORD(TemplateComponentOutputStructure_hwID_out_7.Item2).%B2;
            // _data_out_8[4]                     :=      TO_DWORD(TemplateComponentOutputStructure_hwID_out_7.Item2).%B3;

            _retVal := Siemens.Simatic.DistributedIO.WriteData((Config.HWIDs.HwID_out_7),_data_out_8);
            IF _retVal > WORD#0 THEN
                Messenger.Activate(UINT#1237, eAxoMessageCategory#ProgrammingError);
                Status.Error.Id := UINT#1237;
                RETURN;
            END_IF;

            // _data_out_8[3]                     :=      TO_DWORD(TemplateComponentOutputStructure_hwID_out_8.Item1).%B0;
            // _data_out_8[2]                     :=      TO_DWORD(TemplateComponentOutputStructure_hwID_out_8.Item1).%B1;
            // _data_out_8[1]                     :=      TO_DWORD(TemplateComponentOutputStructure_hwID_out_8.Item1).%B2;
            // _data_out_8[0]                     :=      TO_DWORD(TemplateComponentOutputStructure_hwID_out_8.Item1).%B3;
            // _data_out_8[7]                     :=      TO_DWORD(TemplateComponentOutputStructure_hwID_out_8.Item2).%B0;
            // _data_out_8[6]                     :=      TO_DWORD(TemplateComponentOutputStructure_hwID_out_8.Item2).%B1;
            // _data_out_8[5]                     :=      TO_DWORD(TemplateComponentOutputStructure_hwID_out_8.Item2).%B2;
            // _data_out_8[4]                     :=      TO_DWORD(TemplateComponentOutputStructure_hwID_out_8.Item2).%B3;

            _retVal := Siemens.Simatic.DistributedIO.WriteData((Config.HWIDs.HwID_out_8),_data_out_8);
            IF _retVal > WORD#0 THEN
                Messenger.Activate(UINT#1238, eAxoMessageCategory#ProgrammingError);
                Status.Error.Id := UINT#1238;
                RETURN;
            END_IF;

            // _data_out_8[3]                     :=      TO_DWORD(TemplateComponentOutputStructure_hwID_out_9.Item1).%B0;
            // _data_out_8[2]                     :=      TO_DWORD(TemplateComponentOutputStructure_hwID_out_9.Item1).%B1;
            // _data_out_8[1]                     :=      TO_DWORD(TemplateComponentOutputStructure_hwID_out_9.Item1).%B2;
            // _data_out_8[0]                     :=      TO_DWORD(TemplateComponentOutputStructure_hwID_out_9.Item1).%B3;
            // _data_out_8[7]                     :=      TO_DWORD(TemplateComponentOutputStructure_hwID_out_9.Item2).%B0;
            // _data_out_8[6]                     :=      TO_DWORD(TemplateComponentOutputStructure_hwID_out_9.Item2).%B1;
            // _data_out_8[5]                     :=      TO_DWORD(TemplateComponentOutputStructure_hwID_out_9.Item2).%B2;
            // _data_out_8[4]                     :=      TO_DWORD(TemplateComponentOutputStructure_hwID_out_9.Item2).%B3;

            _retVal := Siemens.Simatic.DistributedIO.WriteData((Config.HWIDs.HwID_out_9),_data_out_8);
            IF _retVal > WORD#0 THEN
                Messenger.Activate(UINT#1239, eAxoMessageCategory#ProgrammingError);
                Status.Error.Id := UINT#1239;
                RETURN;
            END_IF;

            // _data_out_8[3]                     :=      TO_DWORD(TemplateComponentOutputStructure_hwID_out_10.Item1).%B0;
            // _data_out_8[2]                     :=      TO_DWORD(TemplateComponentOutputStructure_hwID_out_10.Item1).%B1;
            // _data_out_8[1]                     :=      TO_DWORD(TemplateComponentOutputStructure_hwID_out_10.Item1).%B2;
            // _data_out_8[0]                     :=      TO_DWORD(TemplateComponentOutputStructure_hwID_out_10.Item1).%B3;
            // _data_out_8[7]                     :=      TO_DWORD(TemplateComponentOutputStructure_hwID_out_10.Item2).%B0;
            // _data_out_8[6]                     :=      TO_DWORD(TemplateComponentOutputStructure_hwID_out_10.Item2).%B1;
            // _data_out_8[5]                     :=      TO_DWORD(TemplateComponentOutputStructure_hwID_out_10.Item2).%B2;
            // _data_out_8[4]                     :=      TO_DWORD(TemplateComponentOutputStructure_hwID_out_10.Item2).%B3;

            _retVal := Siemens.Simatic.DistributedIO.WriteData((Config.HWIDs.HwID_out_10),_data_out_8);
            IF _retVal > WORD#0 THEN
                Messenger.Activate(UINT#1240, eAxoMessageCategory#ProgrammingError);
                Status.Error.Id := UINT#1240;
                RETURN;
            END_IF;

            // _data_out_1[0].%X1                  :=      TemplateComponentOutputStructure_hwID_out_11.Item1;
            // _data_out_1[0].%X2                  :=      TemplateComponentOutputStructure_hwID_out_11.Item2;
            // _data_out_1[0].%X3                  :=      TemplateComponentOutputStructure_hwID_out_11.Item1;
            // _data_out_1[0].%X4                  :=      TemplateComponentOutputStructure_hwID_out_11.Item2;

            _retVal := Siemens.Simatic.DistributedIO.WriteData((Config.HWIDs.HwID_out_11),_data_out_1);
            IF _retVal > WORD#0 THEN
                Messenger.Activate(UINT#1241, eAxoMessageCategory#ProgrammingError);
                Status.Error.Id := UINT#1241;
                RETURN;
            END_IF;

            // _data_out_1[0].%X1                  :=      TemplateComponentOutputStructure_hwID_out_12.Item1;
            // _data_out_1[0].%X2                  :=      TemplateComponentOutputStructure_hwID_out_12.Item2;
            // _data_out_1[0].%X3                  :=      TemplateComponentOutputStructure_hwID_out_12.Item1;
            // _data_out_1[0].%X4                  :=      TemplateComponentOutputStructure_hwID_out_12.Item2;

            _retVal := Siemens.Simatic.DistributedIO.WriteData((Config.HWIDs.HwID_out_12),_data_out_1);
            IF _retVal > WORD#0 THEN
                Messenger.Activate(UINT#1242, eAxoMessageCategory#ProgrammingError);
                Status.Error.Id := UINT#1242;
                RETURN;
            END_IF;

            // _data_out_4[1]                     :=      TO_WORD(TemplateComponentOutputStructure_hwID_out_13.Item1).%B0;
            // _data_out_4[0]                     :=      TO_WORD(TemplateComponentOutputStructure_hwID_out_13.Item1).%B1;
            // _data_out_4[3]                     :=      TO_WORD(TemplateComponentOutputStructure_hwID_out_13.Item2).%B0;
            // _data_out_4[2]                     :=      TO_WORD(TemplateComponentOutputStructure_hwID_out_13.Item2).%B1;

            _retVal := Siemens.Simatic.DistributedIO.WriteData((Config.HWIDs.HwID_out_13),_data_out_4);
            IF _retVal > WORD#0 THEN
                Messenger.Activate(UINT#1243, eAxoMessageCategory#ProgrammingError);
                Status.Error.Id := UINT#1243;
                RETURN;
            END_IF;

            // _data_out_8[3]                     :=      TO_DWORD(TemplateComponentOutputStructure_hwID_out_14.Item1).%B0;
            // _data_out_8[2]                     :=      TO_DWORD(TemplateComponentOutputStructure_hwID_out_14.Item1).%B1;
            // _data_out_8[1]                     :=      TO_DWORD(TemplateComponentOutputStructure_hwID_out_14.Item1).%B2;
            // _data_out_8[0]                     :=      TO_DWORD(TemplateComponentOutputStructure_hwID_out_14.Item1).%B3;
            // _data_out_8[7]                     :=      TO_DWORD(TemplateComponentOutputStructure_hwID_out_14.Item2).%B0;
            // _data_out_8[6]                     :=      TO_DWORD(TemplateComponentOutputStructure_hwID_out_14.Item2).%B1;
            // _data_out_8[5]                     :=      TO_DWORD(TemplateComponentOutputStructure_hwID_out_14.Item2).%B2;
            // _data_out_8[4]                     :=      TO_DWORD(TemplateComponentOutputStructure_hwID_out_14.Item2).%B3;

            _retVal := Siemens.Simatic.DistributedIO.WriteData((Config.HWIDs.HwID_out_14),_data_out_8);
            IF _retVal > WORD#0 THEN
                Messenger.Activate(UINT#1244, eAxoMessageCategory#ProgrammingError);
                Status.Error.Id := UINT#1244;
                RETURN;
            END_IF;

            // _data_out_8[3]                     :=      TO_DWORD(TemplateComponentOutputStructure_hwID_out_15.Item1).%B0;
            // _data_out_8[2]                     :=      TO_DWORD(TemplateComponentOutputStructure_hwID_out_15.Item1).%B1;
            // _data_out_8[1]                     :=      TO_DWORD(TemplateComponentOutputStructure_hwID_out_15.Item1).%B2;
            // _data_out_8[0]                     :=      TO_DWORD(TemplateComponentOutputStructure_hwID_out_15.Item1).%B3;
            // _data_out_8[7]                     :=      TO_DWORD(TemplateComponentOutputStructure_hwID_out_15.Item2).%B0;
            // _data_out_8[6]                     :=      TO_DWORD(TemplateComponentOutputStructure_hwID_out_15.Item2).%B1;
            // _data_out_8[5]                     :=      TO_DWORD(TemplateComponentOutputStructure_hwID_out_15.Item2).%B2;
            // _data_out_8[4]                     :=      TO_DWORD(TemplateComponentOutputStructure_hwID_out_15.Item2).%B3;

            _retVal := Siemens.Simatic.DistributedIO.WriteData((Config.HWIDs.HwID_out_15),_data_out_8);
            IF _retVal > WORD#0 THEN
                Messenger.Activate(UINT#1245, eAxoMessageCategory#ProgrammingError);
                Status.Error.Id := UINT#1245;
                RETURN;
            END_IF;

            // _data_out_8[3]                     :=      TO_DWORD(TemplateComponentOutputStructure_hwID_out_16.Item1).%B0;
            // _data_out_8[2]                     :=      TO_DWORD(TemplateComponentOutputStructure_hwID_out_16.Item1).%B1;
            // _data_out_8[1]                     :=      TO_DWORD(TemplateComponentOutputStructure_hwID_out_16.Item1).%B2;
            // _data_out_8[0]                     :=      TO_DWORD(TemplateComponentOutputStructure_hwID_out_16.Item1).%B3;
            // _data_out_8[7]                     :=      TO_DWORD(TemplateComponentOutputStructure_hwID_out_16.Item2).%B0;
            // _data_out_8[6]                     :=      TO_DWORD(TemplateComponentOutputStructure_hwID_out_16.Item2).%B1;
            // _data_out_8[5]                     :=      TO_DWORD(TemplateComponentOutputStructure_hwID_out_16.Item2).%B2;
            // _data_out_8[4]                     :=      TO_DWORD(TemplateComponentOutputStructure_hwID_out_16.Item2).%B3;

            _retVal := Siemens.Simatic.DistributedIO.WriteData((Config.HWIDs.HwID_out_16),_data_out_8);
            IF _retVal > WORD#0 THEN
                Messenger.Activate(UINT#1246, eAxoMessageCategory#ProgrammingError);
                Status.Error.Id := UINT#1246;
                RETURN;
            END_IF;

            // _data_out_8[3]                     :=      TO_DWORD(TemplateComponentOutputStructure_hwID_out_17.Item1).%B0;
            // _data_out_8[2]                     :=      TO_DWORD(TemplateComponentOutputStructure_hwID_out_17.Item1).%B1;
            // _data_out_8[1]                     :=      TO_DWORD(TemplateComponentOutputStructure_hwID_out_17.Item1).%B2;
            // _data_out_8[0]                     :=      TO_DWORD(TemplateComponentOutputStructure_hwID_out_17.Item1).%B3;
            // _data_out_8[7]                     :=      TO_DWORD(TemplateComponentOutputStructure_hwID_out_17.Item2).%B0;
            // _data_out_8[6]                     :=      TO_DWORD(TemplateComponentOutputStructure_hwID_out_17.Item2).%B1;
            // _data_out_8[5]                     :=      TO_DWORD(TemplateComponentOutputStructure_hwID_out_17.Item2).%B2;
            // _data_out_8[4]                     :=      TO_DWORD(TemplateComponentOutputStructure_hwID_out_17.Item2).%B3;

            _retVal := Siemens.Simatic.DistributedIO.WriteData((Config.HWIDs.HwID_out_17),_data_out_8);
            IF _retVal > WORD#0 THEN
                Messenger.Activate(UINT#1247, eAxoMessageCategory#ProgrammingError);
                Status.Error.Id := UINT#1247;
                RETURN;
            END_IF;

            // _data_out_8[3]                     :=      TO_DWORD(TemplateComponentOutputStructure_hwID_out_18.Item1).%B0;
            // _data_out_8[2]                     :=      TO_DWORD(TemplateComponentOutputStructure_hwID_out_18.Item1).%B1;
            // _data_out_8[1]                     :=      TO_DWORD(TemplateComponentOutputStructure_hwID_out_18.Item1).%B2;
            // _data_out_8[0]                     :=      TO_DWORD(TemplateComponentOutputStructure_hwID_out_18.Item1).%B3;
            // _data_out_8[7]                     :=      TO_DWORD(TemplateComponentOutputStructure_hwID_out_18.Item2).%B0;
            // _data_out_8[6]                     :=      TO_DWORD(TemplateComponentOutputStructure_hwID_out_18.Item2).%B1;
            // _data_out_8[5]                     :=      TO_DWORD(TemplateComponentOutputStructure_hwID_out_18.Item2).%B2;
            // _data_out_8[4]                     :=      TO_DWORD(TemplateComponentOutputStructure_hwID_out_18.Item2).%B3;

            _retVal := Siemens.Simatic.DistributedIO.WriteData((Config.HWIDs.HwID_out_18),_data_out_8);
            IF _retVal > WORD#0 THEN
                Messenger.Activate(UINT#1248, eAxoMessageCategory#ProgrammingError);
                Status.Error.Id := UINT#1248;
                RETURN;
            END_IF;

            // _data_out_8[3]                     :=      TO_DWORD(TemplateComponentOutputStructure_hwID_out_19.Item1).%B0;
            // _data_out_8[2]                     :=      TO_DWORD(TemplateComponentOutputStructure_hwID_out_19.Item1).%B1;
            // _data_out_8[1]                     :=      TO_DWORD(TemplateComponentOutputStructure_hwID_out_19.Item1).%B2;
            // _data_out_8[0]                     :=      TO_DWORD(TemplateComponentOutputStructure_hwID_out_19.Item1).%B3;
            // _data_out_8[7]                     :=      TO_DWORD(TemplateComponentOutputStructure_hwID_out_19.Item2).%B0;
            // _data_out_8[6]                     :=      TO_DWORD(TemplateComponentOutputStructure_hwID_out_19.Item2).%B1;
            // _data_out_8[5]                     :=      TO_DWORD(TemplateComponentOutputStructure_hwID_out_19.Item2).%B2;
            // _data_out_8[4]                     :=      TO_DWORD(TemplateComponentOutputStructure_hwID_out_19.Item2).%B3;

            _retVal := Siemens.Simatic.DistributedIO.WriteData((Config.HWIDs.HwID_out_19),_data_out_8);
            IF _retVal > WORD#0 THEN
                Messenger.Activate(UINT#1249, eAxoMessageCategory#ProgrammingError);
                Status.Error.Id := UINT#1249;
                RETURN;
            END_IF;

            // _data_out_8[3]                     :=      TO_DWORD(TemplateComponentOutputStructure_hwID_out_20.Item1).%B0;
            // _data_out_8[2]                     :=      TO_DWORD(TemplateComponentOutputStructure_hwID_out_20.Item1).%B1;
            // _data_out_8[1]                     :=      TO_DWORD(TemplateComponentOutputStructure_hwID_out_20.Item1).%B2;
            // _data_out_8[0]                     :=      TO_DWORD(TemplateComponentOutputStructure_hwID_out_20.Item1).%B3;
            // _data_out_8[7]                     :=      TO_DWORD(TemplateComponentOutputStructure_hwID_out_20.Item2).%B0;
            // _data_out_8[6]                     :=      TO_DWORD(TemplateComponentOutputStructure_hwID_out_20.Item2).%B1;
            // _data_out_8[5]                     :=      TO_DWORD(TemplateComponentOutputStructure_hwID_out_20.Item2).%B2;
            // _data_out_8[4]                     :=      TO_DWORD(TemplateComponentOutputStructure_hwID_out_20.Item2).%B3;

            _retVal := Siemens.Simatic.DistributedIO.WriteData((Config.HWIDs.HwID_out_20),_data_out_8);
            IF _retVal > WORD#0 THEN
                Messenger.Activate(UINT#1250, eAxoMessageCategory#ProgrammingError);
                Status.Error.Id := UINT#1250;
                RETURN;
            END_IF;

            //******************************************

        END_METHOD

        METHOD PUBLIC TemplateMethod_10steps_1 : IAxoTaskState
            TemplateMethod_10steps_1 := TemplateTask_10steps_1.Invoke(THIS);
        END_METHOD

        METHOD PUBLIC TemplateMethod_10steps_2 : IAxoTaskState
            TemplateMethod_10steps_2 := TemplateTask_10steps_2.Invoke(THIS);
        END_METHOD

        METHOD PUBLIC TemplateMethod_10steps_3 : IAxoTaskState
            TemplateMethod_10steps_3 := TemplateTask_10steps_3.Invoke(THIS);
        END_METHOD

        METHOD PUBLIC TemplateMethod_10steps_4 : IAxoTaskState
            TemplateMethod_10steps_4 := TemplateTask_10steps_4.Invoke(THIS);
        END_METHOD

        METHOD PUBLIC TemplateMethod_10steps_5 : IAxoTaskState
            TemplateMethod_10steps_5 := TemplateTask_10steps_5.Invoke(THIS);
        END_METHOD

        METHOD PUBLIC TemplateMethod_10steps_6 : IAxoTaskState
            TemplateMethod_10steps_6 := TemplateTask_10steps_6.Invoke(THIS);
        END_METHOD

        METHOD PUBLIC TemplateMethod_20steps_1 : IAxoTaskState
            TemplateMethod_20steps_1 := TemplateTask_20steps_1.Invoke(THIS);
        END_METHOD

        METHOD PUBLIC TemplateMethod_20steps_2 : IAxoTaskState
            TemplateMethod_20steps_2 := TemplateTask_20steps_2.Invoke(THIS);
        END_METHOD

        METHOD PUBLIC TemplateMethod_20steps_3 : IAxoTaskState
            TemplateMethod_20steps_3 := TemplateTask_20steps_3.Invoke(THIS);
        END_METHOD

        METHOD PUBLIC TemplateMethod_20steps_4 : IAxoTaskState
            TemplateMethod_20steps_4 := TemplateTask_20steps_4.Invoke(THIS);
        END_METHOD

        METHOD PUBLIC TemplateMethod_20steps_5 : IAxoTaskState
            TemplateMethod_20steps_5 := TemplateTask_20steps_5.Invoke(THIS);
        END_METHOD

        METHOD PUBLIC TemplateMethod_20steps_6 : IAxoTaskState
            TemplateMethod_20steps_6 := TemplateTask_20steps_6.Invoke(THIS);
        END_METHOD

        METHOD PROTECTED OVERRIDE ManualControl
            THIS._isManuallyControllable := true;
        END_METHOD

        ///<summary>
        /// Restores this component into intial state.
        ///</summary>
        METHOD PUBLIC OVERRIDE Restore
            VAR
                _index : INT;
            END_VAR
            Status.Action.Id := UINT#0;
            Status.Error.Id  := UINT#0;

            _progress       :=   INT#0;
            _retVal    :=   WORD#0;

            _data_out_1[0] := BYTE#0;
            _data_out_2[0] := BYTE#0;
            _data_out_2[1] := BYTE#0;

            FOR _index := 0 TO 3 DO
                _data_in[_index] := BYTE#0;
                _data_out_4[_index] := BYTE#0;
                _data_out_8[_index] := BYTE#0;
                _data_out_255[_index] := BYTE#0;
            END_FOR;

            FOR _index := 4 TO 7 DO
                _data_in[_index] := BYTE#0;
                _data_out_8[_index] := BYTE#0;
                _data_out_255[_index] := BYTE#0;
            END_FOR;

            FOR _index := 8 TO 254 DO
                _data_in[_index] := BYTE#0;
                _data_out_255[_index] := BYTE#0;
            END_FOR;

            _word           :=   WORD#0;
            _dword          :=   DWORD#0;

            TemplateTask_10steps_1.Restore();
            TemplateTask_10steps_2.Restore();
            TemplateTask_10steps_3.Restore();
            TemplateTask_10steps_4.Restore();
            TemplateTask_10steps_5.Restore();
            TemplateTask_10steps_6.Restore();
            TemplateTask_20steps_1.Restore();
            TemplateTask_20steps_2.Restore();
            TemplateTask_20steps_3.Restore();
            TemplateTask_20steps_4.Restore();
            TemplateTask_20steps_5.Restore();
            TemplateTask_20steps_6.Restore();
            HardwareDiagnosticsTask.Restore();

            Status.Action.Id := UINT#50;
            RestoreTask.DoneWhen(TRUE);

        END_METHOD

        METHOD PRIVATE CallTimers
            VAR_INPUT
                signal : BOOL;
            END_VAR

            _infoTimer.OnDelay(THIS, signal AND Config.InfoTime > T#0S ,Config.InfoTime);
            _errorTimer.OnDelay(THIS, signal AND Config.ErrorTime > T#0S , Config.ErrorTime);

        END_METHOD

    END_CLASS
END_NAMESPACE
